Staubli VAL3: InstrItem.dtx

public string sType
public string sData
